# EPICS substitutions: ek9000App/Db/EL4028.substitutions
file EL4028.template
{       pattern
        {
                TERMINAL,

        }
        {
        }
}
